// TIA Portal V16 export
// export: Created 2022-11-17T15:49:19.708203Z, ExportSetting WithDefaults, DisplayName Totally Integrated Automation Portal, DisplayVersion V16 Update 6, DisplayName TIA Portal Version Control Interface, DisplayVersion V16 Update 2, DisplayName TIA Portal Openness, DisplayVersion V16 Update 6, DisplayName SINAMICS Startdrive Advanced, DisplayVersion V16 Update 5, DisplayName SINAMICS Startdrive G130, G150, S120, S150, SINAMICS MV, S210, DisplayVersion V16 Update 5, DisplayName SINAMICS Startdrive G110M, G120, G120C, G120D, G120P, G115D, DisplayVersion V16 Update 5, DisplayName STEP 7 Professional, DisplayVersion V16 Update 6, DisplayName STEP 7 Safety, DisplayVersion V16, DisplayName WinCC Advanced, DisplayVersion V16 Update 6
FUNCTION "FC22_NoTop" : Void   // FC22, LAD
TITLE = No top
{ S7_Optimized_Access := 'FALSE' }
AUTHOR : Robopac
VERSION : 0.0
// stored: AutoNumber false, IsIECCheckEnabled false, SetENOAutomatically false, UDAEnableTagReadback false
BEGIN

REGION Network 1: TopOk10: Table rotation middle speed
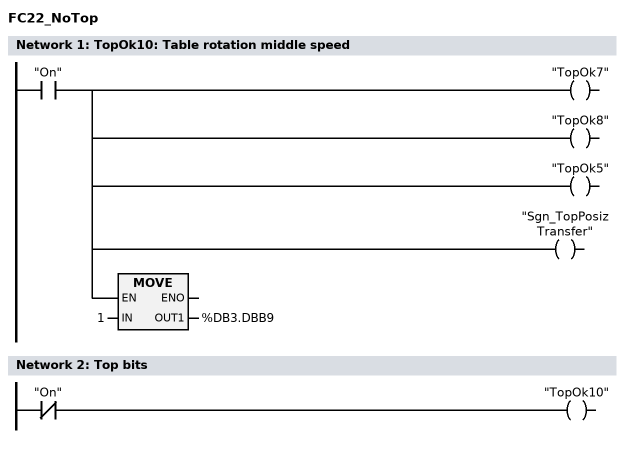
   RUNG wire#powerrail
      Contact( "On" )
      wire#w1
      Coil( "TopOk7" )
   END_RUNG
   RUNG wire#w1
      Coil( "TopOk8" )
   END_RUNG
   RUNG wire#w1
      Coil( "TopOk5" )
   END_RUNG
   RUNG wire#w1
      Coil( "Sgn_TopPosizTransfer" )
   END_RUNG
   RUNG wire#w1
      { S7_GenerateENO := "TRUE" } Move(in := 1, out1 => %DB3.DBB9)
   END_RUNG
   // the same network as SCL:
   "TopOk7" := "On";
   "TopOk8" := "On";
   "TopOk5" := "On";
   "Sgn_TopPosizTransfer" := "On";
   IF "On" THEN %DB3.DBB9 := 1; END_IF;
END_REGION

REGION Network 2: Top bits
   RUNG wire#powerrail
      I_Contact( "On" )
      Coil( "TopOk10" )
   END_RUNG
   // the same network as SCL:
   "TopOk10" := NOT "On";
END_REGION
END_FUNCTION
